(* CODESYS project FsCommon_0.3.1.3.library
   Company: FisoThemes
   DefaultNamespace: FsCommon
   Version: 0.3.1.3
   Placeholder: FsCommon
   Author: Goodwill Mzumala
   Description: A library that contains common utilites and definitiions to streamline and standardise the development of PLC applications.
   Title: FsCommon

Project tree, tasks and I/O mapping:
  libraries: SysTarget, * (System); Tc2_Standard, * (Beckhoff Automation GmbH); Tc2_System, * (Beckhoff Automation GmbH); Tc3_Module, * (Beckhoff Automation GmbH)
  DUTs/
    Primitives/
      data type F32
      data type F64
      data type I16
      data type I32
      data type I64
      data type I8
      data type U16
      data type U32
      data type U64
      data type U8
    data type E_Accessor
    data type E_AddressMemoryArea
    data type E_Comparison
    data type E_OperatingSystem
    data type E_ProcessorArchitecture
    data type T_Char
    data type T_Generic
    data type T_MaxWString
    data type T_PlcAppSysInfo
    data type T_Position
    data type T_QueryInterface
    data type T_Size
    data type T_TaskNameString
    data type T_TypeClass
    data type T_VarInfo
    data type T_WChar
    data type U_Pointer
  GVLs/
    global variables GVL_TypeValueLimits
  ITFs/
    Markers/
    interface I_ChangeDetector: HasChanged
    interface I_Destructable: FB_exit
    interface I_PlcTaskInformation: AdsPort, CycleCount, CycleTime, CycleTimeExceeded, HasCallAfterOutputUpdateAttribute, Index, IsFirstCycle, LastCycleExecutionTime, Name, ObjectId, Priority, RTTimeLimitExceeded
  PARAMs/
  POUs/
    Conversions/
      function F_DintToSize [ST]
      function F_IntToSize [ST]
      function F_PositionToSize [ST]
      function F_SizeToDint [ST]
      function F_SizeToInt [ST]
      function F_SizeToPosition [ST]
      function F_ULintToPosition [ST]
    function F_AllAreFalse [ST]
    function F_AllAreTrue [ST]
    function F_AllocateMemory [ST]
    function F_AnyAreFalse [ST]
    function F_AnyAreTrue [ST]
    function F_DeallocateMemory [ST]
    function F_GetAddressFromInterface [ST]
    function F_GetAddressMemoryArea [ST]
    function F_GetCpuCycleCounter [ST]
    function F_GetCurrentPlcTaskInformation [ST]
    function F_GetInf [ST]
    function F_GetMemorySegment [ST]
    function F_GetNaN [ST]
    function F_GetNumberOfPlcTasks [ST]
    function F_Hash [ST]
    function F_Lerp [ST]
    function F_ResetOnTrue [ST]
    function F_SearchMemory [ST]
    function F_SetDecimalPlaces [ST]
    function F_SwapMemory [ST]
    function block FB_PlcTaskCycleChangeDetector [ST]: CurrentCycle, FB_init, HasChanged, IsFirstCycle, LastCycleChecked, TaskIndex
    function block FB_PlcTaskInformation [ST]: AdsPort, CycleCount, CycleTime, CycleTimeExceeded, FB_init, HasCallAfterOutputUpdateAttribute, Index, IsFirstCycle, LastCycleExecutionTime, Name, ObjectId, Priority, RTTimeLimitExceeded
    function block FB_RandomNumberGenerator [ST]: GetSystemEntropy, LinearCongruentialGenerator, FB_init, NextInt, NextRangedInt, NextRangedReal, NextReal
    function block FB_ValueChangeDetector [ST]: HasChanged
    program P_GetSystemInformation [ST]: CompilerVersion, CompilerVersionNumeric, HasFpuSupport, HasMulticoreSupport, InSimulationMode, IsLittleEndian, OperatingSystem, PackMode, ProcessorArchitecture, RegisterSize, RuntimeVersion, RuntimeVersionNumeric
    program PLAYGROUND [ST]
  Project Information/
    function F_GetCompany [ST]
    function F_GetTitle [ST]
    function F_GetVersion [ST]
  UMLs/
  Version/
    global variables Global_Version
  VISUs/
*)

// DUTs/Primitives/F32
TYPE F32 : REAL; END_TYPE

// DUTs/Primitives/F64
TYPE F64 : LREAL; END_TYPE

// DUTs/Primitives/I16
TYPE I16 : INT; END_TYPE

// DUTs/Primitives/I32
TYPE I32 : DINT; END_TYPE

// DUTs/Primitives/I64
TYPE I64 : LINT; END_TYPE

// DUTs/Primitives/I8
TYPE I8 : SINT; END_TYPE

// DUTs/Primitives/U16
TYPE U16 : UINT; END_TYPE

// DUTs/Primitives/U32
TYPE U32 : UDINT; END_TYPE

// DUTs/Primitives/U64
TYPE U64 : ULINT; END_TYPE

// DUTs/Primitives/U8
TYPE U8 : BYTE; END_TYPE

// DUTs/E_Accessor
// An enum that can be used to represent getters and setters.
{attribute 'qualified_only'}
{attribute 'to_string'}
TYPE E_Accessor :
(
	_ := 0, // Unknown/Invalid
	Get,
	Set
)BYTE;
END_TYPE

// DUTs/E_AddressMemoryArea
// An enum to specify the memory area type of an address.
{attribute 'qualified_only'}
{attribute 'to_string'}
TYPE E_AddressMemoryArea :
(
	_ 		:= 0, 	// Unknown/Invalid.
	Static	:= 1, 	// Static memory.
	Dynamic	:= 2, 	// Dynamic memory.
	CNC		:= 3	// CNC static memory.
)BYTE;
END_TYPE

// DUTs/E_Comparison
// Comparison enum.
{attribute 'qualified_only'}
{attribute 'to_string'}
TYPE E_Comparison :
(
	_ := 0, // Unknown/Invalid
	Less,
	Equal,
	Greater
)BYTE;
END_TYPE

// DUTs/E_OperatingSystem
// Operating system used by the machine.
{attribute 'qualified_only'}
{attribute 'to_string'}
TYPE E_OperatingSystem :
(
	_ 			:= 0, 		// Invalid/Unknown/Ininitialised
	Windows,				// Windows OS
	Linux		:= 5,		// Linux
	VxWorks,				// VxWorks RTOS
	QNX,					// Blackberry QNX Embedded OS
	uCOS					// Micro-Controller Operating Systems by Jean J. Labrosse (1991)
) BYTE;
END_TYPE

// DUTs/E_ProcessorArchitecture
// Processor used by the machine.
{attribute 'qualified_only'}
{attribute 'to_string'}
TYPE E_ProcessorArchitecture :
(
	_ 			:= 0, 	// Invalid/Unknown/Ininitialised
	X86,				// X86 Processor
	ARM,				// ARM Processor
	PowerPC,			// PowerPC Processor
	MIPS				// MIPS processor (as of March 2021 MIPS Technology has moved to RISC-V)
)BYTE;
END_TYPE

// DUTs/T_Char
// Type alias for a single character string.
TYPE T_Char : STRING(1); END_TYPE

// DUTs/T_Generic
// Type alias for a generic type, __SYSTEM.AnyType.
TYPE T_Generic : __SYSTEM.AnyType; END_TYPE

// DUTs/T_MaxWString
// Type alias for a wide string with a maximum length of 255 characters.
TYPE T_MaxWString : WSTRING(255); END_TYPE

// DUTs/T_PlcAppSysInfo
// Type alias for a struct PLC application system information.
TYPE T_PlcAppSysInfo : PlcAppSystemInfo; END_TYPE

// DUTs/T_Position
// Type alias for represeting position.
TYPE T_Position : LINT; END_TYPE

// DUTs/T_QueryInterface
TYPE T_QueryInterface : __SYSTEM.IQueryInterface; END_TYPE

// DUTs/T_Size
// Type alias for represeting size or capacity.
TYPE T_Size : UDINT; END_TYPE

// DUTs/T_TaskNameString
TYPE T_TaskNameString : STRING(63); END_TYPE

// DUTs/T_TypeClass
TYPE T_TypeClass : __SYSTEM.TYPE_CLASS; END_TYPE

// DUTs/T_VarInfo
// Alias for __SYSTEM.VAR_INFO.
// [use] Stores variable information.
TYPE T_VarInfo : __SYSTEM.VAR_INFO; END_TYPE

// DUTs/T_WChar
// Type alias for a single wide character string.
TYPE T_WChar : WSTRING(1); END_TYPE

// DUTs/U_Pointer
// Union to handle various types of pointers in a flexible way.
// This union allows a pointer to be treated as different types, making it versatile for various memory operations.
TYPE U_Pointer :
UNION
	AsPointerToBool			: POINTER TO BOOL;
    AsPointerToByte			: POINTER TO BYTE;
    AsPointerToWord			: POINTER TO WORD;
    AsPointerToDWord		: POINTER TO DWORD;
    AsPointerToLWord		: POINTER TO LWORD;
	AsPointerToXWord		: POINTER TO __XWORD;
    AsPointerToSint			: POINTER TO SINT;
    AsPointerToInt			: POINTER TO INT;
    AsPointerToDint			: POINTER TO DINT;
    AsPointerToLint			: POINTER TO LINT;
	AsPointerToXint			: POINTER TO __XINT;
    AsPointerToUSint		: POINTER TO USINT;
    AsPointerToUInt			: POINTER TO UINT;
    AsPointerToUDint		: POINTER TO UDINT;
    AsPointerToULint		: POINTER TO ULINT;
	AsPointerToUXint		: POINTER TO __UXINT;
    AsPointerToReal			: POINTER TO REAL;
    AsPointerToLReal		: POINTER TO LREAL;
	AsPointerToString		: POINTER TO STRING;
    AsPointerToMaxString	: POINTER TO Tc2_System.T_MaxString;
    AsPointerToWString		: POINTER TO WSTRING;
	AsPointerToMaxWString	: POINTER TO T_MaxWString;
    AsPointerToTime			: POINTER TO TIME;
	AsPointerToLTime 		: POINTER TO LTIME;
    AsPointerToDate			: POINTER TO DATE;
    AsPointerToDateAndTime	: POINTER TO DATE_AND_TIME;
    AsPointerToTimeOfDay	: POINTER TO TIME_OF_DAY;
	AsPointerToInterface 	: POINTER TO __SYSTEM.IQueryInterface;
	AsNestedPointer			: POINTER TO U_Pointer;
	AsVoidPointer			: PVOID;
	AsUnsignedInterger		: __UXINT;
	AsWord					: __XWORD;
END_UNION
END_TYPE

// GVLs/GVL_TypeValueLimits
{attribute 'qualified_only'}
VAR_GLOBAL CONSTANT
    // Minimum and maximum values for BYTE type
    BYTE_MIN        : BYTE           := 0;          // Minimum value for BYTE
    BYTE_MAX        : BYTE           := 255;        // Maximum value for BYTE
    
    // Minimum and maximum values for WORD type
    WORD_MIN        : WORD           := 16#0;       // Minimum value for WORD
    WORD_MAX        : WORD           := 16#FFFF;    // Maximum value for WORD
    
    // Minimum and maximum values for DWORD type
    DWORD_MIN       : DWORD          := 16#0;       // Minimum value for DWORD
    DWORD_MAX       : DWORD          := 16#FFFFFFFF;// Maximum value for DWORD
    
    // Minimum and maximum values for LWORD type
    LWORD_MIN       : LWORD          := 16#0;				 // Minimum value for LWORD
    LWORD_MAX       : LWORD          := 16#FFFFFFFFFFFFFFFF; // Maximum value for LWORD
    
    // Minimum and maximum values for SINT type
    SINT_MIN        : SINT           := -128;       // Minimum value for SINT
    SINT_MAX        : SINT           := +127;       // Maximum value for SINT
    
    // Minimum and maximum values for UINT type
    UINT_MIN        : UINT           := 0;          // Minimum value for UINT
    UINT_MAX        : UINT           := 65535;      // Maximum value for UINT
    
    // Minimum and maximum values for INT type
    INT_MIN         : INT            := -32768;     // Minimum value for INT
    INT_MAX         : INT            := +32767;     // Maximum value for INT
    
    // Minimum and maximum values for UDINT type
    UDINT_MIN       : UDINT          := 0;				// Minimum value for UDINT
    UDINT_MAX       : UDINT          := 4_294_967_295; 	// Maximum value for UDINT
    
    // Minimum and maximum values for DINT type
    DINT_MIN        : DINT           := -2_147_483_648; // Minimum value for DINT
    DINT_MAX        : DINT           := +2_147_483_647; // Maximum value for DINT
    
    // Minimum and maximum values for ULINT type
    ULINT_MIN       : ULINT          := 0;							// Minimum value for ULINT
    ULINT_MAX       : ULINT          := 18_446_744_073_709_551_615; // Maximum value for ULINT
    
    // Minimum and maximum values for LINT type
    LINT_MIN        : LINT           := -9_223_372_036_854_775_808; // Minimum value for LINT
    LINT_MAX        : LINT           := +9_223_372_036_854_775_807; // Maximum value for LINT
    
    // Minimum and maximum values for REAL type
    REAL_MIN        : REAL           := -3.402823E+38; // Minimum value for REAL
    REAL_MAX        : REAL           := +3.402823E+38; // Maximum value for REAL
    
    // Minimum and maximum values for LREAL type
    LREAL_MIN       : LREAL          := -1.7976931348623158E+308; // Minimum value for LREAL
    LREAL_MAX       : LREAL          := +1.7976931348623158E+308; // Maximum value for LREAL
    
    // Minimum and maximum values for TIME type
    TIME_MIN        : TIME           := T#0S;       // Minimum value for TIME
    TIME_MAX        : TIME           := T#49D17H2M47S295MS; // Maximum value for TIME
    
    // Minimum and maximum values for LTIME type
    LTIME_MIN       : LTIME          := LTIME#0S;   // Minimum value for LTIME
    LTIME_MAX       : LTIME          := LTIME#213503D23H34M33S709MS551US615NS; // Maximum value for LTIME
    
    // Minimum and maximum values for DATE type
    DATE_MIN        : DATE           := D#1970-01-01; // Minimum value for DATE
    DATE_MAX        : DATE           := D#2106-02-07; // Maximum value for DATE
    
    // Minimum and maximum values for DT (DateTime) type
    DT_MIN          : DT             := DT#1970-1-1-0:0:0; // Minimum value for DT
    DT_MAX          : DT             := DT#2106-02-07-06:28:15; // Maximum value for DT
    
    // Minimum and maximum values for TOD (Time of Day) type
    TOD_MIN         : TOD            := TOD#0:0:0; // Minimum value for TOD
    TOD_MAX         : TOD            := TOD#23:59:59.999; // Maximum value for TOD
    
    // Minimum and maximum values for T_Size type
    T_SIZE_MIN      : T_Size         := UDINT_MIN;  // Minimum value for T_Size
    T_SIZE_MAX      : T_Size         := UDINT_MAX;  // Maximum value for T_Size
    
    // Minimum and maximum values for T_Position type
    T_POSITION_MIN  : T_Position     := LINT_MIN;   // Minimum value for T_Position
    T_POSITION_MAX  : T_Position     := LINT_MAX;   // Maximum value for T_Position
END_VAR

// Version/Global_Version
{attribute 'TcGenerated'}
{attribute 'no-analysis'}
{attribute 'linkalways'}
// This function has been automatically generated from the project information.
VAR_GLOBAL CONSTANT
	{attribute 'const_non_replaced'}
	stLibVersion_FsCommon : ST_LibVersion := (iMajor := 0, iMinor := 3, iBuild := 1, iRevision := 3, nFlags := 0, sVersion := '0.3.1.3');
END_VAR

// ITFs/I_ChangeDetector
// Interface for indicating that an object is for detecting the change of some object/value.
INTERFACE I_ChangeDetector EXTENDS __SYSTEM.IQueryInterface

// Indicates if the object has changed.
// [get] Returns flag indicating of object has changed.
PROPERTY HasChanged : BOOL
GET
END_GET
END_PROPERTY

END_INTERFACE

// ITFs/I_Destructable
// Interface to indicate that an object has resources that need to be released.
INTERFACE I_Destructable EXTENDS __SYSTEM.IQueryInterface

METHOD FB_exit : BOOL
VAR_INPUT
	bInCopyCode : BOOL; // if TRUE, the exit method is called for exiting an instance that is copied afterwards (online change).
END_VAR
END_METHOD

END_INTERFACE

// ITFs/I_PlcTaskInformation
// Interface for accessing information about a PLC task.
INTERFACE I_PlcTaskInformation EXTENDS __SYSTEM.IQueryInterface

// Task's ADS Port.
// [get] Returns the referenced task's ADS port.
PROPERTY AdsPort : UINT
GET
END_GET
END_PROPERTY

// The task's cycle counter.
// [note] This refers to the actual system task and not to the task reference of the PLC project.
// [get] Returns the task's cycle counter.
PROPERTY CycleCount : UDINT
GET
END_GET
END_PROPERTY

// The cycle time of the task.
// [get] Returns the cycle time.
PROPERTY CycleTime : LTIME
GET
END_GET
END_PROPERTY

// Indicates whether the cycle time has been exceeded.
// [get] Returns TRUE if the cycle time has been exceeded.
PROPERTY CycleTimeExceeded : BOOL
GET
END_GET
END_PROPERTY

// Indicates if the origin of the current call is declared with the attribute 'TcCallAfterOutputUpdate'.
// [get] Returns TRUE if current call is declared with the attribute 'TcCallAfterOutputUpdate'.
PROPERTY HasCallAfterOutputUpdateAttribute : BOOL
GET
END_GET
END_PROPERTY

// The index of the task.
// [get] Returns the index.
PROPERTY Index : DINT
GET
END_GET
END_PROPERTY

// Indicates if it is the first cycle of the task.
// [get] Returns TRUE if it is the first cycle.
PROPERTY IsFirstCycle : BOOL
GET
END_GET
END_PROPERTY

// Time the previous cycle took to complete execution.
// [get] Returns the last exection time.
PROPERTY LastCycleExecutionTime : LTIME
GET
END_GET
END_PROPERTY

// The name of the task.
// [get] Returns the task name.
PROPERTY Name : T_TaskNameString
GET
END_GET
END_PROPERTY

// The object ID of the task reference, from which the PLC program is called.
// [get] Returns the object ID.
PROPERTY ObjectId : OTCID
GET
END_GET
END_PROPERTY

// The priority of the task.
// [get] Returns the priority.
PROPERTY Priority : UINT
GET
END_GET
END_PROPERTY

// Indicates whether the real-time time limit has been exceeded on a mixed core (Windows + real-time on one core).
// [get] Returns true if the real-time time limit has been exceeded.
PROPERTY RTTimeLimitExceeded : BOOL
GET
END_GET
END_PROPERTY

END_INTERFACE

// POUs/Conversions/F_DintToSize
// Converts a DINT value to a size value, ensuring it falls within the defined limits.
FUNCTION F_DintToSize : T_Size // The size value constrained within the minimum and maximum limits of T_Size.
VAR_INPUT
	nValue : DINT; // The DINT value to be converted to a size value.
END_VAR
VAR
END_VAR

F_DintToSize := TO_UDINT(
	LIMIT(0, nValue, GVL_TypeValueLimits.DINT_MAX));

END_FUNCTION

// POUs/Conversions/F_IntToSize
// Converts a INT value to a size value, ensuring it falls within the defined limits.
FUNCTION F_IntToSize : T_Size // The size value constrained within the minimum and maximum limits of T_Size.
VAR_INPUT
	nValue : INT; // The INT value to be converted to a size value.
END_VAR
VAR
END_VAR

F_IntToSize := TO_UDINT(
	LIMIT(0, nValue, GVL_TypeValueLimits.INT_MAX));

END_FUNCTION

// POUs/Conversions/F_PositionToSize
// Converts a position value to a size value, ensuring it falls within the defined limits.
FUNCTION F_PositionToSize : T_Size // The size value corresponding to the given position, constrained within the minimum and maximum limits of T_Size.
VAR_INPUT
	Position : T_Position; // The position value to be converted to a size value.
END_VAR

F_PositionToSize := TO_UDINT(
	LIMIT(
		GVL_TypeValueLimits.T_SIZE_MIN, 
		Position, 
		GVL_TypeValueLimits.T_SIZE_MAX));

END_FUNCTION

// POUs/Conversions/F_SizeToDint
// Converts a T_Size value to a DINT value.
FUNCTION F_SizeToDint : DINT // The converted DINT value from the given T_Size.
VAR_INPUT
	Size : T_Size; // The input size to be converted.
END_VAR

F_SizeToDint := TO_DINT(LIMIT(0, Size, TO_UDINT(GVL_TypeValueLimits.DINT_MAX)));

END_FUNCTION

// POUs/Conversions/F_SizeToInt
// Converts a T_Size value to a INT value.
FUNCTION F_SizeToInt : INT // The converted INT value from the given T_Size.
VAR_INPUT
	Size : T_Size; // The input size to be converted.
END_VAR

F_SizeToInt := TO_INT(LIMIT(0, Size, TO_UDINT(GVL_TypeValueLimits.INT_MAX)));

END_FUNCTION

// POUs/Conversions/F_SizeToPosition
// Converts a size value to a position value.
FUNCTION F_SizeToPosition : T_Position // The position value corresponding to the given size.
VAR_INPUT
	Size : T_Size; // The size value to be converted to a position value.
END_VAR

F_SizeToPosition := Size;

END_FUNCTION

// POUs/Conversions/F_ULintToPosition
// Converts a ULINT value to a position value, ensuring it falls within the defined limits.
FUNCTION F_ULintToPosition : T_Position // The position value constrained within the minimum and maximum limits of T_Position.
VAR_INPUT
	nValue : ULINT; // The size value to be converted to a position value.
END_VAR

F_ULintToPosition := TO_LINT(LIMIT(0, nValue, TO_ULINT(GVL_TypeValueLimits.LINT_MAX)));

END_FUNCTION

// POUs/F_AllAreFalse
// Checks if all elements in a boolean array are false.
FUNCTION F_AllAreFalse : BOOL // True if all elements in the array are false.
VAR_IN_OUT
	arValues : ARRAY[*] OF BOOL; // An array of boolean values to check.
END_VAR
VAR
	i : T_Position;
END_VAR

FOR i := LOWER_BOUND(arValues, 1) TO UPPER_BOUND(arValues, 1) DO
	IF arValues[i] THEN RETURN; END_IF 
	END_FOR
	
F_AllAreFalse := TRUE;

END_FUNCTION

// POUs/F_AllAreTrue
// Checks if all elements in a boolean array are true.
FUNCTION F_AllAreTrue : BOOL // True if all elements in the array are true.
VAR_IN_OUT
	arValues : ARRAY[*] OF BOOL; // An array of boolean values to check.
END_VAR
VAR
	i : T_Position;
END_VAR

FOR i := LOWER_BOUND(arValues, 1) TO UPPER_BOUND(arValues, 1) DO
	IF NOT arValues[i] THEN RETURN; END_IF 
	END_FOR
	
F_AllAreTrue := TRUE;

END_FUNCTION

// POUs/F_AllocateMemory
// Allocates a block of dynamic memory of the specified size.
FUNCTION F_AllocateMemory : POINTER TO BYTE // A pointer to the beginning of the newly allocated memory block.
VAR_INPUT
	Size : T_Size; // The size, in bytes, of the memory block to be allocated.
END_VAR

F_AllocateMemory := __NEW(BYTE, Size);

END_FUNCTION

// POUs/F_AnyAreFalse
// Checks if any element in a boolean array is false.
FUNCTION F_AnyAreFalse : BOOL // True if any element in the array is false.
VAR_IN_OUT
	arValues : ARRAY[*] OF BOOL; // An array of boolean values to check.
END_VAR
VAR
	i : T_Position;
END_VAR

FOR i := LOWER_BOUND(arValues, 1) TO UPPER_BOUND(arValues, 1) DO
	IF NOT arValues[i] THEN F_AnyAreFalse := TRUE; RETURN; END_IF 
	END_FOR

END_FUNCTION

// POUs/F_AnyAreTrue
// Checks if any element in a boolean array is true.
FUNCTION F_AnyAreTrue : BOOL // True if any element in the array is true.
VAR_IN_OUT
	arValues : ARRAY[*] OF BOOL; // An array of boolean values to check.
END_VAR
VAR
	i : T_Position;
END_VAR

FOR i := LOWER_BOUND(arValues, 1) TO UPPER_BOUND(arValues, 1) DO
	IF arValues[i] THEN F_AnyAreTrue := TRUE; RETURN; END_IF 
	END_FOR

END_FUNCTION

// POUs/F_DeallocateMemory
// Safely releases a memory pointer. 
// Ensuring that dynamically allocated memory is properly deallocated,
// and statically allocated memory pointers are safely nullified to avoid potential memory issues.
FUNCTION F_DeallocateMemory
VAR_IN_OUT
	pAddress : POINTER TO BYTE; // The memory pointer to be released.
END_VAR

IF NOT __ISVALIDREF(pAddress) THEN RETURN; END_IF

CASE Tc2_System.F_CheckMemoryArea(pAddress, 1) OF
	Tc2_System.E_TcMemoryArea.Dynamic:
		__DELETE(pAddress); 
ELSE
	pAddress := 0;
	END_CASE

END_FUNCTION

// POUs/F_GetAddressFromInterface
// Retrieves the memory address of an object given its interface.
FUNCTION F_GetAddressFromInterface : POINTER TO BYTE // A pointer to the memory address of the object corresponding to the provided interface pointer.
VAR_INPUT
	ipInterface : __SYSTEM.IQueryInterface; // The interface from which the address of the object will be extracted.
END_VAR
VAR
	pInterface : POINTER TO POINTER TO BYTE := ADR(ipInterface);
END_VAR

F_GetAddressFromInterface := SEL(ipInterface <> 0, 0, pInterface^ - SIZEOF(ipInterface));

END_FUNCTION

// POUs/F_GetAddressMemoryArea
// Determines the memory area type of a given pointer.
FUNCTION F_GetAddressMemoryArea : E_AddressMemoryArea // An enumeration indicating the type of memory area the address belongs to.
VAR_INPUT
	pAddress : POINTER TO BYTE; // The memory address pointer to be checked.
END_VAR

CASE Tc2_System.F_CheckMemoryArea(pAddress, 1) OF
	Tc2_System.E_TcMemoryArea.Static:	F_GetAddressMemoryArea := E_AddressMemoryArea.Static;
	Tc2_System.E_TcMemoryArea.Dynamic:	F_GetAddressMemoryArea := E_AddressMemoryArea.Dynamic;
	Tc2_System.E_TcMemoryArea.CNC:		F_GetAddressMemoryArea := E_AddressMemoryArea.CNC;
ELSE
	F_GetAddressMemoryArea := E_AddressMemoryArea._;
	END_CASE

END_FUNCTION

// POUs/F_GetCpuCycleCounter
// Gets the CPU's cycle count.
// The value us refreshed every 100ns.
FUNCTION F_GetCpuCycleCounter : ULINT // The current CPU count with in the 100ns refresh rate.
VAR_STAT
	fbGetCpuCounter : Tc2_System.GETCPUCOUNTER;
END_VAR

fbGetCpuCounter();
F_GetCpuCycleCounter := SHL(TO_ULINT(fbGetCpuCounter.cpuCntHiDW), 32) OR fbGetCpuCounter.cpuCntLoDW;

END_FUNCTION

// POUs/F_GetCurrentPlcTaskInformation
// Retrieves the information about the current PLC task.
FUNCTION F_GetCurrentPlcTaskInformation : I_PlcTaskInformation // An instance of I_PlcTaskInformation containing details of the current PLC task.
VAR_STAT
	fbGetCurrentTaskIndex : Tc2_System.GETCURTASKINDEX;
	fbPlcTaskInformation : FB_PlcTaskInformation;
END_VAR

fbGetCurrentTaskIndex();
fbPlcTaskInformation.Index 		:= fbGetCurrentTaskIndex.Index;
F_GetCurrentPlcTaskInformation 	:= fbPlcTaskInformation;

END_FUNCTION

// POUs/FB_PlcTaskInformation
// Retrieves PLC Task information.
// [note] if not explicitly defined, the default task index is the task the function block is instatiated on. 
{attribute 'enable_dynamic_creation'}
{attribute 'no_explicit_call' := 'direct call for this function block is not allowed'}
FUNCTION_BLOCK FINAL FB_PlcTaskInformation IMPLEMENTS I_PlcTaskInformation
VAR
	_nTaskIndex : DINT;
END_VAR

// Task's ADS Port.
// [get] Returns the referenced task's ADS port.
PROPERTY AdsPort : Tc2_System.T_AmsPort
GET
AdsPort := TwinCAT_SystemInfoVarList._TaskInfo[THIS^._nTaskIndex].AdsPort;
END_GET
END_PROPERTY

// The task's cycle counter.
// [note] This refers to the actual system task and not to the task reference of the PLC project.
// [get] Returns the task's cycle counter.
PROPERTY CycleCount : UDINT
GET
CycleCount := TwinCAT_SystemInfoVarList._TaskInfo[THIS^._nTaskIndex].CycleCount;
END_GET
END_PROPERTY

// The cycle time of the task.
// [get] Returns the cycle time.
PROPERTY CycleTime : LTIME
GET
CycleTime := TO_LTIME(TwinCAT_SystemInfoVarList._TaskInfo[THIS^._nTaskIndex].CycleTime * 100);
END_GET
END_PROPERTY

// Indicates whether the cycle time has been exceeded.
// [get] Returns TRUE if the cycle time has been exceeded.
PROPERTY CycleTimeExceeded : BOOL
GET
CycleTimeExceeded := TwinCAT_SystemInfoVarList._TaskInfo[THIS^._nTaskIndex].CycleTimeExceeded;
END_GET
END_PROPERTY

{attribute 'hide'}
METHOD FB_init : BOOL
VAR_INPUT
	bInitRetains : BOOL; // if TRUE, the retain variables are initialized (warm start / cold start)
	bInCopyCode : BOOL;  // if TRUE, the instance afterwards gets moved into the copy code (online change)
END_VAR
VAR
	fbGetCurrentTaskIndex : Tc2_System.GETCURTASKINDEX;
END_VAR
fbGetCurrentTaskIndex(Index => THIS^._nTaskIndex);
END_METHOD

// Indicates if the origin of the current call is declared with the attribute 'TcCallAfterOutputUpdate'.
// [get] Returns TRUE if current call is declared with the attribute 'TcCallAfterOutputUpdate'.
PROPERTY HasCallAfterOutputUpdateAttribute : BOOL
GET
HasCallAfterOutputUpdateAttribute := TwinCAT_SystemInfoVarList._TaskInfo[THIS^._nTaskIndex].InCallAfterOutputUpdate;
END_GET
END_PROPERTY

// The index of the task.
// [get] Returns the index.
// [set] The index of the task to retrieve information from.
PROPERTY Index : DINT
GET
Index := THIS^._nTaskIndex;
END_GET
SET
THIS^._nTaskIndex := LIMIT(1, Index, F_SizeToDint(F_GetNumberOfPlcTasks()));
END_SET
END_PROPERTY

// Indicates if it is the first cycle of the task.
// [get] Returns TRUE if it is the first cycle.
PROPERTY IsFirstCycle : BOOL
GET
IsFirstCycle := TwinCAT_SystemInfoVarList._TaskInfo[THIS^._nTaskIndex].FirstCycle;
END_GET
END_PROPERTY

// Time the previous cycle took to complete execution.
// [get] Returns the last exection time.
PROPERTY LastCycleExecutionTime : LTIME
GET
LastCycleExecutionTime := TO_LTIME(TwinCAT_SystemInfoVarList._TaskInfo[THIS^._nTaskIndex].LastExecTime * 100);
END_GET
END_PROPERTY

// The name of the task.
// [get] Returns the task name.
PROPERTY Name : T_TaskNameString
GET
Name := TwinCAT_SystemInfoVarList._TaskInfo[THIS^._nTaskIndex].TaskName;
END_GET
END_PROPERTY

// The object ID of the task reference, from which the PLC program is called.
// [get] Returns the object ID.
PROPERTY ObjectId : OTCID
GET
ObjectId := TwinCAT_SystemInfoVarList._TaskInfo[THIS^._nTaskIndex].ObjId;
END_GET
END_PROPERTY

// The priority of the task.
// [get] Returns the priority.
PROPERTY Priority : UINT
GET
Priority := TwinCAT_SystemInfoVarList._TaskInfo[THIS^._nTaskIndex].Priority;
END_GET
END_PROPERTY

// Indicates whether the real-time time limit has been exceeded on a mixed core (Windows + real-time on one core).
// [get] Returns true if the real-time time limit has been exceeded.
PROPERTY RTTimeLimitExceeded : BOOL
GET
RTTimeLimitExceeded := TwinCAT_SystemInfoVarList._TaskInfo[THIS^._nTaskIndex].RTViolation;
END_GET
END_PROPERTY

END_FUNCTION_BLOCK

// POUs/F_GetNumberOfPlcTasks
// Retrieves the number of PLC tasks available in the system.
FUNCTION F_GetNumberOfPlcTasks : T_Size // The number of PLC tasks.

F_GetNumberOfPlcTasks := SIZEOF(TwinCAT_SystemInfoVarList._TaskInfo) / SIZEOF(PlcTaskSystemInfo);

END_FUNCTION

// POUs/F_GetInf
// Retrieves the positive infinity value for LREAL data type.
FUNCTION F_GetInf : LREAL // The positive infinity value.
VAR_STAT
	fInf : LREAL := TO_LREAL('#Inf');
END_VAR

F_GetInf := fInf;

END_FUNCTION

// POUs/F_GetMemorySegment
//	Retrieves the memory address of a segment of memory.
FUNCTION F_GetMemorySegment : POINTER TO BYTE // A pointer to the memory location of the specified segment.
VAR_INPUT
    pAddress : POINTER TO BYTE; // Starting address of the memory location.
    Size     : T_Size; // Size of one segment.
    Index    : T_Position; // Index of the segment.
END_VAR

F_GetMemorySegment := SEL(pAddress <> 0, 0, pAddress + (Size * F_PositionToSize(Index)));

END_FUNCTION

// POUs/F_GetNaN
// Retrieves the "Not-a-Number" (NaN) value for LREAL data type.
FUNCTION F_GetNaN : LREAL // The NaN value.
VAR_STAT
	fNaN : LREAL := TO_LREAL('#NaN');
END_VAR

F_GetNaN := fNaN;

END_FUNCTION

// POUs/F_Hash
// Computes a hash value for a given block of memory using the MurmurHash3 algorithm.
// The MurmurHash3 algorithm was created by Austin Appleby. Source: https://en.wikipedia.org/wiki/MurmurHash
FUNCTION F_Hash : DWORD // The computed hash value.
VAR_INPUT
    pAddress 	: POINTER TO BYTE; // The pointer to the beginning of the memory block to be hashed.
    Size 		: T_Size; // The size, in bytes, of the memory block to be hashed.
    Seed 		: DWORD; // A seed value for the hash calculation, which can help in generating different hashes for the same data.
END_VAR
VAR
	i 			: T_Position;
	nK 			: DWORD;
	nBlocks 	: T_Size;
	pBlocks		: POINTER TO DWORD;
	pTail 		: POINTER TO BYTE;
END_VAR
VAR_STAT CONSTANT
	nC1 		: DWORD 			:= 16#CC9E2D51;
	nC2 		: DWORD 			:= 16#1B873593;
END_VAR

IF pAddress = 0 OR Size = 0 THEN RETURN; END_IF

F_Hash := Seed;

nBlocks := Size / 4;
pBlocks := pAddress + nBlocks * 4;

i := -F_SizeToPosition(nBlocks);
FOR i := i TO -1 DO
	nK := pBlocks[i];
	
	nK := nK * nC1;
	nK := SHL(nK, 15) OR SHR(nK, 32 - 15);
	nK := nK * nC2;
	
	F_Hash := F_Hash XOR nK;
	F_Hash := SHL(F_Hash, 13) OR SHR(F_Hash, 32 - 13);
	F_Hash := F_Hash * 5 + 16#E6546B64;
	END_FOR
	
nK := 0;
pTail := pAddress + nBlocks * 4;

i := Size MOD 4;

IF i = 3 THEN 
	{warning disable C0308}
	nK := nK XOR SHL(pTail[2], 16); END_IF;
IF i >= 2 THEN 
	{warning disable C0308}	
	nK := nK XOR SHL(pTail[1], 8); END_IF;
IF i >= 1 THEN
	nK := nK XOR pTail[0];
	nK := nK * nC1;
	nK := SHL(nK, 15) OR SHR(nK, 32 - 15);
	nK := nK * nC2;
	F_Hash := F_Hash XOR nK;
	END_IF;

F_Hash := F_Hash XOR Size;
F_Hash := F_Hash XOR SHR(F_Hash, 16);
F_Hash := F_Hash * 16#85EBCA6B;
F_Hash := F_Hash XOR SHR(F_Hash, 13);
F_Hash := F_Hash * 16#C2B2AE35;
F_Hash := F_Hash XOR SHR(F_Hash, 16);

END_FUNCTION

// POUs/F_Lerp
// Linearly interpolates between two values based on a given percentage.
FUNCTION F_Lerp : LREAL // The interpolated value.
VAR_INPUT
    fStartValue : LREAL; // The starting value.
    fEndValue   : LREAL; // The ending value.
    fPercentage : LREAL; // The interpolation factor (0.0 to 1.0).
END_VAR

F_Lerp := fStartValue + (fEndValue - fStartValue) * fPercentage;

END_FUNCTION

// POUs/F_ResetOnTrue
// Sets the boolean value to false if it is true and returns true if it was true before being set.
FUNCTION F_ResetOnTrue : BOOL // Whether the value was true before resetting.
VAR_INPUT
	bValue : REFERENCE TO BOOL; // Boolean value to reset.
END_VAR

IF bValue THEN bValue := FALSE; F_ResetOnTrue := TRUE; END_IF

END_FUNCTION

// POUs/F_SearchMemory
// Searches for a specific sequence of bytes in a given memory area.
FUNCTION F_SearchMemory : POINTER TO BYTE // Pointer to the start of the found sequence, or 0 if not found.
VAR_INPUT
    pAddress    : POINTER TO BYTE; // Starting address of the memory area to search.
    Size 		: T_Size; // Size of the memory area (in bytes).
    pValue   	: POINTER TO BYTE; // Pointer to the sequence of bytes to search for.
    ValueSize	: T_Size; // Size of the sequence of bytes (in bytes).
END_VAR
VAR_OUTPUT
	Index		: T_Position := -1; // Index of the start of the found sequence, or -1 if not found.
END_VAR
VAR
    i, j,
	iEnd, jEnd	: T_Position;
END_VAR

IF pAddress = 0 OR pValue = 0 OR ValueSize = 0 THEN RETURN; END_IF

iEnd := F_SizeToPosition(Size) - ValueSize;
jEnd := F_SizeToPosition(ValueSize) - 1;
FOR i := 0 TO iEnd DO
	FOR j := 0 TO jEnd DO
		IF pAddress[i + j] <> pValue[j] THEN EXIT; END_IF
		END_FOR
	IF j = ValueSize THEN F_SearchMemory := ADR(pAddress[i]); Index := j; RETURN; END_IF
	END_FOR

END_FUNCTION

// POUs/F_SetDecimalPlaces
// Sets the specified number of decimal places for a given real value.
FUNCTION F_SetDecimalPlaces : LREAL // The value rounded to the specified number of decimal places.
VAR_INPUT
	fValue 			: LREAL; // The input floating-point value to be rounded.
	nDecimalPlaces 	: USINT; // The number of decimal places to round to.
END_VAR

F_SetDecimalPlaces := TO_DINT(fValue * EXPT(10, nDecimalPlaces)) / EXPT(10, nDecimalPlaces);

END_FUNCTION

// POUs/F_SwapMemory
// Swaps the contents of two memory locations.
FUNCTION F_SwapMemory
VAR_INPUT
    pAddress1 	: POINTER TO BYTE; // Pointer to the first memory location.
    pAddress2 	: POINTER TO BYTE; // Pointer to the second memory location.
    Size 		: T_Size;          // Size of each memory element (in bytes).
END_VAR
VAR
	i, End 			: T_Position;
	nTmp 			: __XWORD;
	pTmpAddress1	: POINTER TO __XWORD := pAddress1;	
	pTmpAddress2	: POINTER TO __XWORD := pAddress2;
END_VAR

IF pAddress1 = pAddress2 OR pAddress1 = 0 OR pAddress2 = 0 THEN RETURN; END_IF

End := TO_LINT(Size / SIZEOF(__XWORD)) - 1;
FOR i := 0 TO End DO
	nTmp := pTmpAddress1[i];
	pTmpAddress1[i] := pTmpAddress2[i];
	pTmpAddress2[i] := nTmp;
	END_FOR

End := TO_LINT(Size) - 1;
FOR i := i TO End DO
	nTmp := pAddress1[i];
	pAddress1[i] := pAddress2[i];
	pAddress2[i] := TO_BYTE(nTmp);
	END_FOR

END_FUNCTION

// POUs/FB_PlcTaskCycleChangeDetector
// Detects if the current PLC task cycle has changed.
// If index of the initialiser less than 1, the task index the object is instatiated on is watched.
// [init] <Instance Name> : FB_PlcTaskCycleChangeDetector(<Task Index>);
{attribute 'enable_dynamic_creation'}
{attribute 'no_explicit_call' := 'direct call for this function block is not allowed'}
FUNCTION_BLOCK FINAL FB_PlcTaskCycleChangeDetector IMPLEMENTS I_ChangeDetector
VAR
	_nTaskIndex 		: DINT	:= 1;
	_nLastCycleChecked 	: UDINT := GVL_TypeValueLimits.UDINT_MAX; // The last cycle checked for change-in-plc-cycle.
END_VAR

// The task's current cycle counter.
// [note] This refers to the actual system task and not to the task reference of the PLC project.
// [get] Returns the current task's cycle counter.
PROPERTY CurrentCycle : UDINT
GET
CurrentCycle := TwinCAT_SystemInfoVarList._TaskInfo[THIS^._nTaskIndex].CycleCount;
END_GET
END_PROPERTY

{attribute 'hide'}
METHOD FB_init : BOOL
VAR_INPUT
	bInitRetains 	: BOOL; // if TRUE, the retain variables are initialized (warm start / cold start)
	bInCopyCode 	: BOOL; // if TRUE, the instance afterwards gets moved into the copy code (online change)
	nTaskIndex 		: DINT; // Index of task to monitor. 0 or less = Task the object is instatiated at.
END_VAR
THIS^._nTaskIndex := SEL(nTaskIndex > 0,
						 F_GetCurrentPlcTaskInformation().Index,
						 LIMIT(1, nTaskIndex, F_SizeToDint(F_GetNumberOfPlcTasks())));
END_METHOD

// Indicates if the value has changed.
// [get] Returns flag indicating of value has changed.
PROPERTY HasChanged : BOOL
GET
HasChanged := THIS^.CurrentCycle <> THIS^._nLastCycleChecked;
THIS^._nLastCycleChecked := THIS^.CurrentCycle;
END_GET
END_PROPERTY

// Indicates if it is the first cycle of the task.
// [get] Returns TRUE if it is the first cycle.
PROPERTY IsFirstCycle : BOOL
GET
 IsFirstCycle := TwinCAT_SystemInfoVarList._TaskInfo[THIS^._nTaskIndex].FirstCycle;
END_GET
END_PROPERTY

// The last cycle checked for change-in-plc-cycle.
// [get] Returns the last cycle checked.
PROPERTY LastCycleChecked : UDINT
GET
LastCycleChecked := THIS^._nLastCycleChecked;
END_GET
END_PROPERTY

// The index of the task being monitored.
// [get] Returns the index.
PROPERTY TaskIndex : DINT
GET
TaskIndex := THIS^._nTaskIndex;
END_GET
END_PROPERTY

END_FUNCTION_BLOCK

// POUs/FB_RandomNumberGenerator
// Generates pseudo-random numbers.
// [init] <Instance Name> : FB_RandomNumberGenerator(<Initial Seed>);
// [note] The methods in this function block can be called using ADS-RPC.
{attribute 'enable_dynamic_creation'}
{attribute 'no_explicit_call' := 'direct call for this function block is not allowed'}
FUNCTION_BLOCK FINAL FB_RandomNumberGenerator IMPLEMENTS __SYSTEM.IQueryInterface
VAR
	_nSeed : LINT;
END_VAR
VAR_STAT CONSTANT
	_nLGC_M : LINT := LINT#9223372036854775783;
END_VAR

// Generates additional entropy based on system timestamp, task time and CPU cycle.
METHOD PRIVATE GetSystemEntropy : LINT // System entropy.
VAR_INPUT
	nSeed : LINT;
END_VAR
GetSystemEntropy := TO_LINT(TO_ULINT(nSeed) XOR Tc2_System.F_GetSystemTime() XOR Tc2_System.F_GetTaskTime() XOR F_GetCpuCycleCounter());
END_METHOD

// LCG formula for updating the seed.
METHOD PRIVATE LinearCongruentialGenerator : LINT // New seed value.
VAR_INPUT
	nSeed : LINT;
END_VAR
LinearCongruentialGenerator := (LINT#6364136223846793005 * nSeed * LINT#1442695040888963407) MOD THIS^._nLGC_M;
END_METHOD

{attribute 'hide'}
METHOD FB_init : BOOL
VAR_INPUT
	bInitRetains 	: BOOL; // if TRUE, the retain variables are initialized (warm start / cold start)
	bInCopyCode 	: BOOL; // if TRUE, the instance afterwards gets moved into the copy code (online change)
	nSeed 			: LINT; // Initial seed value for the generator.
END_VAR
THIS^._nSeed := nSeed;
END_METHOD

// Generates the next pseudo-random integer.
{attribute 'TcRpcEnable'}
METHOD NextInt : LINT // The next pseudo-random integer.
VAR_INPUT
END_VAR
NextInt := THIS^._nSeed := THIS^.LinearCongruentialGenerator(TO_LINT(TO_ULINT(THIS^._nSeed) XOR TO_ULINT(THIS^.GetSystemEntropy(THIS^._nSeed))));
END_METHOD

// Generates the next pseudo-random integer within the specified range [minimum, maximum].
{attribute 'TcRpcEnable'}
METHOD NextRangedInt : LINT // The next pseudo-random integer within the range.
VAR_INPUT
	nMinimum : LINT; // Minimum value of the range. 
	nMaximum : LINT; // Maximum value of the range.
END_VAR
NextRangedInt := MIN(nMinimum, nMaximum) + (ABS(THIS^.NextInt()) MOD (MAX(nMinimum, nMaximum) - MIN(nMinimum, nMaximum) + 1));
END_METHOD

// Generates the next pseudo-random real number within the specified range [minimum, maximum].
{attribute 'TcRpcEnable'}
METHOD NextRangedReal : LREAL // The next pseudo-random real number within the range.
VAR_INPUT
	fMinimum : LREAL; // Minimum value of the range. 
	fMaximum : LREAL; // Maximum value of the range.
END_VAR
NextRangedReal := MIN(fMinimum, fMaximum) + (ABS(THIS^.NextReal()) * (MAX(fMinimum, fMaximum) - MIN(fMinimum, fMaximum)));
END_METHOD

// Generates the next pseudo-random real number.
{attribute 'TcRpcEnable'}
METHOD NextReal : LREAL // The next pseudo-random real number.
VAR_INPUT
END_VAR
NextReal := TO_LREAL(THIS^.NextInt()) / TO_LREAL(THIS^._nLGC_M + 1);
END_METHOD

END_FUNCTION_BLOCK

// POUs/FB_ValueChangeDetector
// Detects if the watched variable value has changed.
{attribute 'enable_dynamic_creation'}
FUNCTION_BLOCK FINAL FB_ValueChangeDetector IMPLEMENTS I_ChangeDetector
VAR_INPUT
	Value : ANY; // Value to detect for change.
END_VAR
VAR
	_nHash : DWORD;
END_VAR

// Indicates if the value has changed.
// [get] Returns flag indicating of value has changed.
PROPERTY HasChanged : BOOL
GET
VAR_INST
	bFirstCall : BOOL := TRUE;
END_VAR
VAR
	nHash : DWORD;
END_VAR
nHash := F_Hash(THIS^.Value.pValue,
				F_PositionToSize(THIS^.Value.diSize),
				THIS^.Value.TypeClass);

HasChanged := THIS^._nHash <> nHash OR_ELSE F_ResetOnTrue(bFirstCall);

IF HasChanged THEN THIS^._nHash := nHash; END_IF
END_GET
END_PROPERTY

END_FUNCTION_BLOCK

// POUs/P_GetSystemInformation
// Retrieves information about the target.
{attribute 'no_explicit_call' := 'direct call for this program is not allowed'} 
PROGRAM P_GetSystemInformation

// The version as defined in the compile options.
PROPERTY CompilerVersion : VERSION
GET
CompilerVersion := __SYSTEM.Constants.CompilerVersion;
END_GET
END_PROPERTY

// The version as defined in the compile options.
PROPERTY CompilerVersionNumeric : DWORD
GET
CompilerVersionNumeric := __SYSTEM.Constants.CompilerVersionNumeric;
END_GET
END_PROPERTY

// Indicates of whether the target has FPU support.
PROPERTY HasFpuSupport : BOOL
GET
HasFpuSupport := __SYSTEM.Constants.bFPUSupport;
END_GET
END_PROPERTY

// Indicates whether multicore support is available in the target.
PROPERTY HasMulticoreSupport : BOOL
GET
HasMulticoreSupport := __SYSTEM.Constants.bMulticoreSupport;
END_GET
END_PROPERTY

// Indicates if target is in simulation mode.
PROPERTY InSimulationMode : BOOL
GET
InSimulationMode := __SYSTEM.Constants.bSimulationMode;
END_GET
END_PROPERTY

// Indicates of the system is little endian; TRUE for Intel, ARM etc. FALSE for Power PC, etc. 
PROPERTY IsLittleEndian : BOOL
GET
IsLittleEndian := __SYSTEM.Constants.bLittleEndian;
END_GET
END_PROPERTY

// Retrieves the operating system of the target.
PROPERTY OperatingSystem : E_OperatingSystem
GET
VAR_STAT
	nOperatingSystem : UDINT;
	nResult : UDINT := SysTarget.SysTargetGetOperatingSystemId(ADR(nOperatingSystem));
END_VAR
CASE nOperatingSystem OF
	1..4: OperatingSystem := E_OperatingSystem.Windows;
	5: OperatingSystem := E_OperatingSystem.Linux;
	6: OperatingSystem := E_OperatingSystem.VxWorks;
	7: OperatingSystem := E_OperatingSystem.QNX;
	8: OperatingSystem := E_OperatingSystem.uCOS;
ELSE
	OperatingSystem := E_OperatingSystem._;
	END_CASE
END_GET
END_PROPERTY

// Retrieves the packmode of the system.
PROPERTY PackMode : WORD
GET
PackMode := __SYSTEM.Constants.nPackMode;
END_GET
END_PROPERTY

// Retireves the target's processor architecture.
PROPERTY ProcessorArchitecture : E_ProcessorArchitecture
GET
VAR_STAT
	nProcessorArchitecture : UDINT;
	nResult : UDINT := SysTarget.SysTargetGetProcessorId(ADR(nProcessorArchitecture));
END_VAR
ProcessorArchitecture := TO_BYTE(nProcessorArchitecture);
END_GET
END_PROPERTY

// Retrieves the size of the CPU register; 16 for C16x, 64 for X86-64 Bit, 32 for all other controllers.
PROPERTY RegisterSize : WORD
GET
RegisterSize := __SYSTEM.Constants.nRegisterSize;
END_GET
END_PROPERTY

// The version as described in the runtime system.
PROPERTY RuntimeVersion : VERSION
GET
RuntimeVersion := __SYSTEM.Constants.RuntimeVersion;
END_GET
END_PROPERTY

// The version as described in the runtime system.
PROPERTY RuntimeVersionNumeric : DWORD
GET
RuntimeVersionNumeric := __SYSTEM.Constants.RuntimeVersionNumeric;
END_GET
END_PROPERTY

END_PROGRAM

// POUs/PLAYGROUND
{attribute 'no_explicit_call' := 'direct call for this program is not allowed'} 
PROGRAM INTERNAL PLAYGROUND
VAR
	Str1, Str2				: T_MaxString;
	pFound 					: POINTER TO STRING;
	uPointer 				: U_Pointer := (AsPointerToString := ADR(Str1));
	bStart 					: BOOL := TRUE;
	nCpuCycle				: ULINT;
	eOpSys 					: E_OperatingSystem;
	eProcArc				: E_ProcessorArchitecture;
	ipTaskInfo 				: I_PlcTaskInformation;
	fbTaskInfo 				: FB_PlcTaskInformation;
	fbTaskCycleChanged		: FB_PlcTaskCycleChangeDetector(0); 
	nHash 					: DWORD;
	AmsPort 				: Tc2_System.T_AmsPort;
	CycleTime, LastExecTime : LTIME;
	i, j, Count, Size 		: T_Size;
	Str 					: STRING := '123456789';
	fbGenRand				: FB_RandomNumberGenerator(0);
	nRand1, nRand2			: LINT;
	fRand1, fRand2			: LREAL;
END_VAR

nHash := F_Hash(ADR(Str), F_PositionToSize(LEN(Str)), 0);

nCpuCycle		:= F_GetCpuCycleCounter();
eProcArc 		:= P_GetSystemInformation.ProcessorArchitecture;
eOpSys 			:= P_GetSystemInformation.OperatingSystem;
AmsPort 		:= F_GetCurrentPlcTaskInformation().AdsPort;
CycleTime 		:= F_GetCurrentPlcTaskInformation().CycleTime;
LastExecTime 	:= F_GetCurrentPlcTaskInformation().LastCycleExecutionTime;
Count 			:= F_GetCurrentPlcTaskInformation().CycleCount;
Size 			:= F_GetNumberOfPlcTasks();

nRand1 := fbGenRand.NextInt();
nRand2 := fbGenRand.NextRangedInt(10, -10);
fRand1 := fbGenRand.NextReal();
fRand2 := F_SetDecimalPlaces(fbGenRand.NextRangedReal(-5.8, 9.432), 2);

pFound := F_SearchMemory(ADR(Str1), F_IntToSize(LEN(Str1)), ADR(Str2), F_IntToSize(LEN(Str2)));

IF NOT F_ResetOnTrue(bStart) THEN RETURN; END_IF

i := SEL(fbTaskCycleChanged.HasChanged, i, i + 1);
j := SEL(fbTaskCycleChanged.HasChanged, j, j + 1);

END_PROGRAM

// Project Information/F_GetCompany
// This function has been automatically generated from the project information.
{attribute 'signature_flag' := '1073741824'}
{attribute 'TcGenerated'}
{attribute 'no-analysis'}
FUNCTION F_GetCompany : WSTRING
VAR_INPUT
	
END_VAR

F_GetCompany := "FisoThemes";

END_FUNCTION

// Project Information/F_GetTitle
// This function has been automatically generated from the project information.
{attribute 'signature_flag' := '1073741824'}
{attribute 'TcGenerated'}
{attribute 'no-analysis'}
FUNCTION F_GetTitle : WSTRING
VAR_INPUT
	
END_VAR

F_GetTitle := "FsCommon";

END_FUNCTION

// Project Information/F_GetVersion
// This function has been automatically generated from the project information.
{attribute 'signature_flag' := '1073741824'}
{attribute 'TcGenerated'}
{attribute 'no-analysis'}
FUNCTION F_GetVersion : ST_LibVersion
VAR_INPUT
	
END_VAR

F_GetVersion.iMajor := 0;
F_GetVersion.iMinor := 3;
F_GetVersion.iBuild := 1;
F_GetVersion.iRevision := 3;

END_FUNCTION
